(* PLC project Generated.project, CODESYS CODESYS V3.5 SP19 Patch 1 *)
(* stored: creationDateTime 2026-09-06T13:00:42.474667, modificationDateTime 2026-09-06T13:00:42.474667 *)

(* values of E_WinchTraceBlockReason: NONE: Aucun blocage - au moins un sens effectivement permis; POWER_CUTOFF: Coupure puissance amont (instSafetyWinch.PowerCutOff) - priorite max; AXIS_DISABLED: Axe neutralise (Mode=DISABLE ou InhibitMx -> Enable FALSE); SAFESTOP: SafeStop effectif (rampe rapide demandee); SAFETY_FAULT: Defaut safety latched (FB_Safety_Winch.Fault.Error); SAFETY_PERMIT_MISSING: Aucun sens ne delivre de permit safety (limite / mou de cable / homing); PROCESS_PERMIT_MISSING: Permit process absent (benne / fond Kobold / limite legale / extraction); COUPLING_BLOCKED: Couplage synchro anti-telescopage (l'autre axe bloque); WINCH_FAULT: Defaut treuil latched (FB_Winch.Fault.Error); FINAL_INTERLOCK_BLOCKED: Barriere finale en defaut (frein / redemarrage) *)

{attribute 'qualified_only'}
{attribute 'strict'}
TYPE E_WinchTraceBlockReason : (NONE := 0, POWER_CUTOFF := 1, AXIS_DISABLED := 2, SAFESTOP := 3, SAFETY_FAULT := 4, SAFETY_PERMIT_MISSING := 5, PROCESS_PERMIT_MISSING := 6, COUPLING_BLOCKED := 7, WINCH_FAULT := 8, FINAL_INTERLOCK_BLOCKED := 9);
END_TYPE
